FUNCTION_BLOCK a2 (* Basic FB with empty ECC *)
  (* Standard: 61499-2 *)
  (* Version 1.0, 2025-03-31, 06220625900 *)
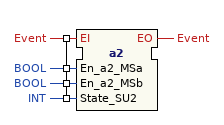
  EVENT_INPUT
    EI WITH En_a2_MSa, En_a2_MSb, State_SU2;
  END_EVENT
  EVENT_OUTPUT
    EO;
  END_EVENT
  VAR_INPUT
    En_a2_MSa : BOOL := False;
    En_a2_MSb : BOOL := False;
    State_SU2 : INT := 1;
  END_VAR
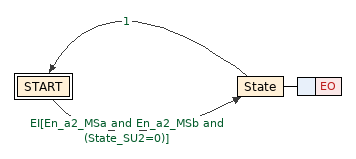
  EC_STATES
    START; (* Initial State *)
    State : -> EO;
  END_STATES
  EC_TRANSITIONS
    START TO State := EI[En_a2_MSa and En_a2_MSb and (State_SU2=0)];
    State TO START := 1;
  END_TRANSITIONS
END_FUNCTION_BLOCK
